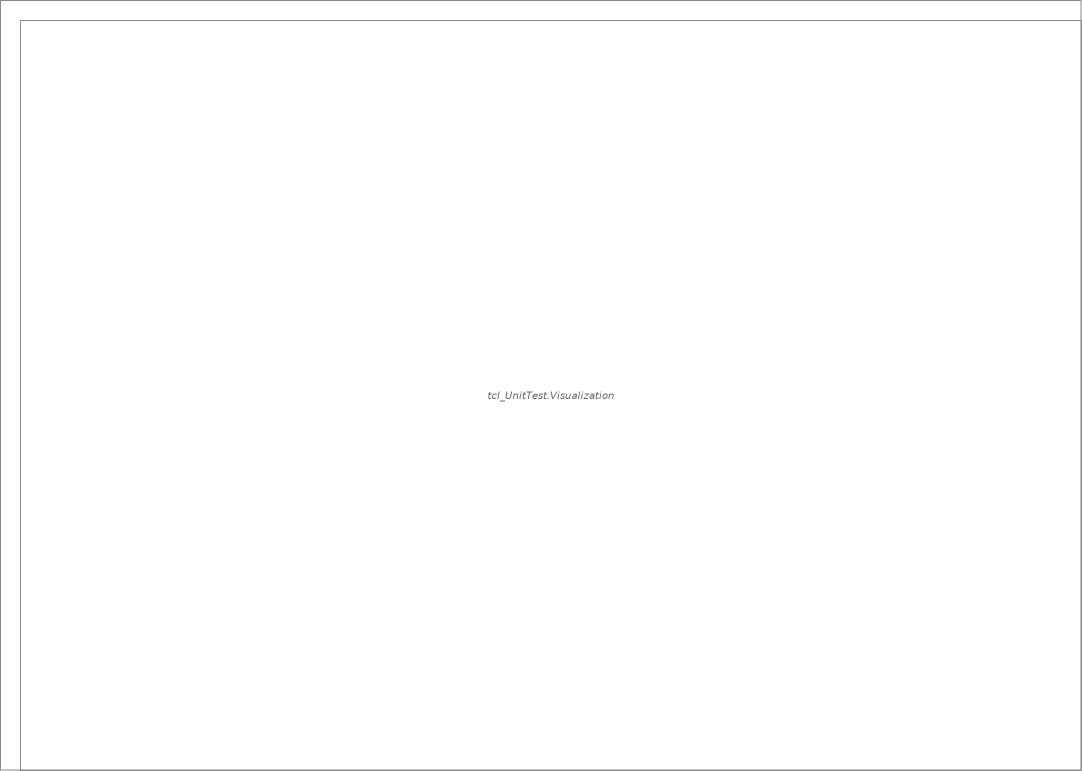
VISUALIZATION Visualization  // 1082x771
    Frame (20,20 1062x751)
        shows tcl_UnitTest.Visualization()
END_VISUALIZATION

(* stored: Version 1.1.0.1, ProductVersion 3.1.4024.3
   Visu Visualization: Id {63d9eeee-e240-07d3-14cf-1ff58e772a61} *)
